TYPE st_BMS_Params :
STRUCT
	IP_BMS							:	STRING(16) := '192.168.1.60';
	r_SocHysteresis					:   REAL := 1; // % 
	r_InternalConditioningSoCMin	: 	REAL := 30;
	r_SoCAbsoluteMin				: 	REAL := 6; // unscaled value
	r_SoCAbsoluteMax				: 	REAL := 100; //unscaled value

	r_KwhperString					: REAL := 208; //
	r_CrateBattery					: REAL := 0.5; //C
	r_AhperString					: REAL := 306; //Ah	
	b_DisableSOCAlarm				: BOOL := FALSE;
	b_ResetPersistentVars			: BOOL := FALSE;
	b_forcePrecharging				: BOOL := FALSE;
	
	b_EnableAutoCalibration			: BOOL := TRUE;
	t_AutoCalibrationInterval 		: TIME := T#14D;
END_STRUCT
END_TYPE

(* stored: Version 1.1.0.1, ProductVersion 3.1.4026.18
   DUT st_BMS_Params: Id {60c5bfe9-7595-4abd-90ef-e9945cabb399} *)
